{attribute addProperty BoxType "EL3681-0000-0021"}
{attribute addProperty Id "SAI_InputsAT %I*SAI_Inputs_166EE3574860SAI_FeedbackAT %I*SAI_Feedback_DF9848341620SAI_RangeAT %Q*SAI_Range_80D0ED7D1620WcStateAT %I*WcState_98A4DF7520.250InfoDataAT %I*InfoData_BC63D37F80100"}
{attribute addProperty CRC "3398425776"}
{attribute addProperty SizeInBites "162"}
{attribute addProperty SizeInBytes "20.25"}
TYPE EL3681_AB553B50 :
STRUCT
	{attribute addProperty Name "SAI_Inputs"}
	SAI_Inputs : SAI_Inputs_166EE357;
	{attribute addProperty Name "SAI_Feedback"}
	SAI_Feedback : SAI_Feedback_DF984834;
	{attribute addProperty Name "SAI_Range"}
	SAI_Range : SAI_Range_80D0ED7D;
	{attribute addProperty Name "WcState"}
	WcState : WcState_98A4DF75;
	{attribute addProperty Name "InfoData"}
	InfoData : InfoData_BC63D37F;
END_STRUCT
END_TYPE

(* stored: Version 1.2.0.0, ProductVersion 3.1.4024.9
   DUT EL3681_AB553B50: Id {0303d1b9-217b-40e6-824d-a10745ee168f} *)
